    M_CROSSCONTROL : UINT := 1624; (* Manufacturer: CrossControl | Location: Alfta, Sweden - 2026-01-27 *)
    M_DMX_POWER : UINT := 1625; (* Manufacturer: DMX Power LLC | Location: Oakdale, MN, USA - 2026-01-27 *)
    M_SMP_STABIL : UINT := 1626; (* Manufacturer: SMP STABIL GmbH | Location: Pécel, Hungary - 2026-01-27 *)
    M_ROTER_ITALIA : UINT := 1627; (* Manufacturer: Roter Italia | Location: Ostiglia(MN), Italy - 2026-01-27 *)
    M_VANEMAR : UINT := 1628; (* Manufacturer: Vanemar, Inc. | Location: Fort Lauderdale, FL, USA - 2026-01-27 *)
    M_DSPACE_SE_AND : UINT := 1629; (* Manufacturer: dSPACE SE & Co. KG | Location: Paderborn, North Rhine Westphalia, Germany - *)
    M_RAINER_MEYER_LANDMASCHINEN : UINT := 1630; (* Manufacturer: Rainer Meyer Landmaschinen GmbH | Location: Niedersachsen, Germany - 2026-01-27 *)
    M_LEIDOS : UINT := 1631; (* Manufacturer: Leidos | Location: Reston, VA, USA - 2026-01-27 *)
    M_ZOCON : UINT := 1632; (* Manufacturer: Zocon | Location: Joure, The Netherlands - 2026-02-09 *)
    M_ZYDRO_MARINE_TECHNOLOGIES : UINT := 1633; (* Manufacturer: Zydro Marine Technologies, Inc. | Location: Boston, MA, USA - 2026-02-09 *)
    M_IBISUL_ELETR_NICA_LTDA : UINT := 1634; (* Manufacturer: IBISUL ELETRÔNICA LTDA | Location: Ibirubá, Rio Grande do Sul, Brazil - 2026-02-09 *)
    M_SAFRAMAX_INDUSTRIAL : UINT := 1635; (* Manufacturer: Saframax Industrial | Location: Campo Mourão, Paraná, Brazil - 2026-02-09 *)
    M_TBB_POWER : UINT := 1636; (* Manufacturer: TBB POWER (XIAMEN) Co., Ltd. | Location: Xiamen, Fujian, China - 2026-02-13 *)
    M_SCHERZINGER_PUMPEN_AND : UINT := 1637; (* Manufacturer: Scherzinger Pumpen GmbH & Co. KG | Location: Furtwangen im Schwarzwald, *)
    M_TEMPA_TEKNIK : UINT := 1638; (* Manufacturer: TEMPA TEKNIK | Location: Tekirdag, Turkey - 2026-02-18 *)
    M_GEA_FARM_TECHNOLOGIES_CANADA : UINT := 1639; (* Manufacturer: GEA Farm Technologies Canada Inc. | Location: Drummondville, QC, Canada - *)
    M_SHANGHAI_INFIPAX_TECHNOLOGY : UINT := 1650; (* Manufacturer: Shanghai Infipax Technology Co., Ltd. | Location: Shanghai, China - 2026-04-03 *)
    M_SCHAFFER_FARMING_TECHNOLOGIES : UINT := 1653; (* Manufacturer: Schaffer Farming Technologies | Location: Mercer, PA, USA - 2026-04-03 *)
    M_SEASTAR_SOLUTIONS : UINT := 1850; (* Manufacturer: Seastar Solutions (formerly Teleflex) | Location: Litchfield, IL - 2021-08-26 *)
    M_RAYMARINE : UINT := 1851; (* Manufacturer: RayMarine | Location: Portsmouth, Hampshire UK - 2003-07-20 *)
    M_NAVIONICS : UINT := 1852; (* Manufacturer: Navionics | Location: Wareham, MA USA - 2003-07-20 *)
    M_JAPAN_RADIO : UINT := 1853; (* Manufacturer: Japan Radio Co | Location: Seattle, WA USA - 2003-07-20 *)
    M_NORTHSTAR_TECHNOLOGIES : UINT := 1854; (* Manufacturer: Northstar Technologies | Location: Acton, MA USA - 2003-07-20 *)
    M_FURUNO_USA : UINT := 1855; (* Manufacturer: Furuno USA | Location: Camas, WA USA - 2003-07-20 *)
    M_TRIMBLE : UINT := 1856; (* Manufacturer: Trimble | Location: Sunnyvale, CA USA - 2003-07-20 *)
    M_SIMRAD : UINT := 1857; (* Manufacturer: Simrad | Location: Egersund, Norway - 2003-07-20 *)
    M_LITTON : UINT := 1858; (* Manufacturer: Litton | Location: Charlottesville, VA USA - 2003-07-20 *)
    M_KVASAR : UINT := 1859; (* Manufacturer: Kvasar AB | Location: Kinnahult, Sweden - 2003-07-20 *)
    M_MMP : UINT := 1860; (* Manufacturer: MMP | Location: Fircrest, WA USA - 2003-07-20 *)
    M_VECTOR_NORTH_AMERICA : UINT := 1861; (* Manufacturer: Vector North America (formerly Vector Cantech) | Location: Novi, MI USA - *)
    M_SANSHIN : UINT := 1862; (* Manufacturer: Sanshin | Location: Shizuoka, Japan - 2003-07-20 *)
    M_THOMAS_G_FARIA : UINT := 1863; (* Manufacturer: Thomas G. Faria Co. | Location: Uncasville, CT USA - 2003-07-20 *)
  END_VAR
END_GLOBALCONSTANTS
